{attribute 'qualified_only'}
{attribute 'strict'}
TYPE E_NOTT_CRYO_CTRL_CMD :
(
	NONE	:= 0,
	COOL,
	WARM_UP
);
END_TYPE

(* stored: Version 1.1.0.1, ProductVersion 3.1.4026.18
   DUT E_NOTT_CRYO_CTRL_CMD: Id {83219e50-94ed-4d54-afc2-12f1385196f1} *)
